ADAPTER TEST_ADP (* Adapter Interface for Testing *)
  (* Standard: 61499-1 *)
  (* Version 0.2, 2005-02-18, JHC, Holobloc Inc, Moved from "student" to "doc". *)
  (* Version 0.1, 2003-08-17, JHC, Rockwell Automation, Moved from "book" to "student". *)
  (* Version 0.0, 2002-01-08, JHC, Rockwell Automation, Built from NEWADAPTER. *)
  (* Compiler header: package fb.rt.doc; *)
  (* Compiler Java IBM Jikes 1.06 *)
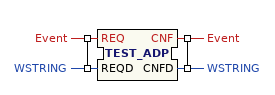
  EVENT_INPUT
    REQ WITH REQD; (* Request from Socket *)
  END_EVENT
  EVENT_OUTPUT
    CNF WITH CNFD; (* Confirmation from Plug *)
  END_EVENT
  VAR_INPUT
    REQD : WSTRING; (* Request Data from Socket *)
  END_VAR
  VAR_OUTPUT
    CNFD : WSTRING; (* Confirmation Data from Plug *)
  END_VAR
  SERVICE SOCKET/PLUG
    SEQUENCE request_confirm
      SOCKET.REQ(REQD) -> PLUG.REQ(REQD);
      PLUG.CNF(CNFD) -> SOCKET.CNF(CNFD);
    END_SEQUENCE
  END_SERVICE
END_ADAPTER
